// TIA Portal V20 export
DATA_BLOCK "SP508"   // DB342
// stored: MemoryReserve 100
   VAR
      "ANODE ALIGN VISION BUSY (STO)" : Bool := FALSE;
      "ANODE ALIGN VISION RESULT (OK)" : Bool := TRUE;
      "STACK VISION BUSY (STO)" : Bool := FALSE;
      "STACK VISION RESULT (OK)" : Bool := FALSE;
      "CATHODE ALIGN VISION BUSY (STO)" : Bool := FALSE;
      "CATHODE ALIGN VISION RESULT (OK)" : Bool := FALSE;
   END_VAR
BEGIN
END_DATA_BLOCK
